// TIA Portal V17 export
FUNCTION "电机启停" : Void   // FC, LAD
{ S7_Optimized_Access := 'TRUE' }
VERSION : 0.1
// stored: AutoNumber true, IsIECCheckEnabled false, SetENOAutomatically false
BEGIN

REGION Network 1
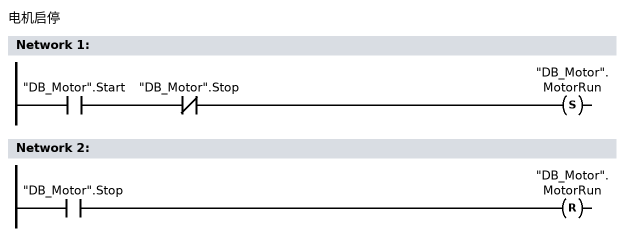
   RUNG wire#powerrail
      Contact( "DB_Motor".Start )
      I_Contact( "DB_Motor".Stop )
      S_Coil( "DB_Motor".MotorRun )
   END_RUNG
   // the same network as SCL:
   IF "DB_Motor".Start AND NOT "DB_Motor".Stop THEN "DB_Motor".MotorRun := TRUE; END_IF;
END_REGION

REGION Network 2
   RUNG wire#powerrail
      Contact( "DB_Motor".Stop )
      R_Coil( "DB_Motor".MotorRun )
   END_RUNG
   // the same network as SCL:
   IF "DB_Motor".Stop THEN "DB_Motor".MotorRun := FALSE; END_IF;
END_REGION
END_FUNCTION
